ORGANIZATION_BLOCK "Startup"
TITLE = "Complete Restart"
{ S7_Optimized_Access := 'TRUE' }
VERSION : 0.1

BEGIN
	"DB_System".firstCycle := TRUE;
END_ORGANIZATION_BLOCK

